# EPICS autosave request: urRobotApp/Db/waypointL_settings.req
$(P)WaypointL:$(N).VAL
$(P)WaypointL:$(N):X.VAL
$(P)WaypointL:$(N):Y.VAL
$(P)WaypointL:$(N):Z.VAL
$(P)WaypointL:$(N):Roll.VAL
$(P)WaypointL:$(N):Pitch.VAL
$(P)WaypointL:$(N):Yaw.VAL
$(P)WaypointL:$(N):Speed.VAL
$(P)WaypointL:$(N):Acceleration.VAL
$(P)WaypointL:$(N):Blend.VAL
$(P)WaypointL:$(N):Enabled
$(P)WaypointL:$(N):ActionOpt
